{attribute 'linkalways'} 
{attribute 'no_explicit_call' := 'This FB is a CLASS and must be accessed using methods or properties'}
{attribute 'enable_dynamic_creation'}
FUNCTION_BLOCK FINAL MIN_UDINT EXTENDS Node
VAR
	in1 : _UDINT(0);
	in2 : _UDINT(0);
	out : _UDINT(0);
END_VAR

METHOD PUBLIC Clone : I_Node
VAR
	pNode : POINTER TO MIN_UDINT;
END_VAR
pNode := __NEW(MIN_UDINT);
Clone := pNode^;
END_METHOD

METHOD FB_init : BOOL
VAR_INPUT
	bInitRetains : BOOL; // if TRUE, the retain variables are initialized (warm start / cold start)
	bInCopyCode : BOOL;  // if TRUE, the instance afterwards gets moved into the copy code (online change)
END_VAR
AddInput('in1',THIS^.in1);
AddInput('in2',THIS^.in2);
AddOutput('out', THIS^.out);
END_METHOD

METHOD PROTECTED OnExecute
VAR
END_VAR
out.Value := MIN(in1.Value, in2.Value);
END_METHOD

END_FUNCTION_BLOCK

(* stored: Version 1.1.0.1, ProductVersion 3.1.4024.15
   POU MIN_UDINT: Id {a28badc3-6324-485c-990b-5e84dc1ebcc3}, SpecialFunc None
   Folder Constructor: Id {6c9178fe-8aee-4db9-8429-60e654e9d7d3}
   Method Clone: Id {1e312733-26a9-4c2a-a854-5a5089aa0c64}
   Method FB_init: Id {a687b971-658a-4040-9ee3-784909a3638f}
   Method OnExecute: Id {905a24a3-7b19-4925-8445-f092fe755197} *)
